// Mitsubishi GX Works2 project: SEMAFARO   PLC: Q03UDV

PROGRAM MAIN
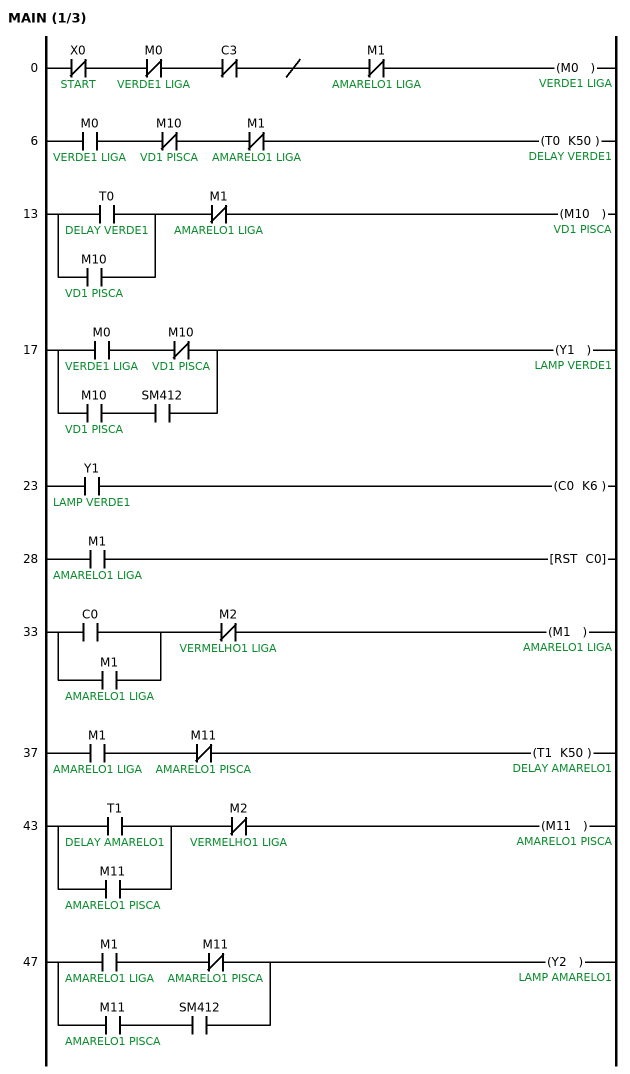
0     LDI     X0  ; START
      ANI     M0  ; VERDE1 LIGA
      ANI     C3
      INV
      ANI     M1  ; AMARELO1 LIGA
      OUT     M0  ; VERDE1 LIGA
6     LD      M0  ; VERDE1 LIGA
      ANI     M10  ; VD1 PISCA
      ANI     M1  ; AMARELO1 LIGA
      OUT     T0 K50  ; DELAY VERDE1
13    LD      T0  ; DELAY VERDE1
      OR      M10  ; VD1 PISCA
      ANI     M1  ; AMARELO1 LIGA
      OUT     M10  ; VD1 PISCA
17    LD      M0  ; VERDE1 LIGA
      ANI     M10  ; VD1 PISCA
      LD      M10  ; VD1 PISCA
      AND     SM412
      ORB
      OUT     Y1  ; LAMP VERDE1
23    LD      Y1  ; LAMP VERDE1
      OUT     C0 K6
28    LD      M1  ; AMARELO1 LIGA
      RST     C0
33    LD      C0
      OR      M1  ; AMARELO1 LIGA
      ANI     M2  ; VERMELHO1 LIGA
      OUT     M1  ; AMARELO1 LIGA
37    LD      M1  ; AMARELO1 LIGA
      ANI     M11  ; AMARELO1 PISCA
      OUT     T1 K50  ; DELAY AMARELO1
43    LD      T1  ; DELAY AMARELO1
      OR      M11  ; AMARELO1 PISCA
      ANI     M2  ; VERMELHO1 LIGA
      OUT     M11  ; AMARELO1 PISCA
47    LD      M1  ; AMARELO1 LIGA
      ANI     M11  ; AMARELO1 PISCA
      LD      M11  ; AMARELO1 PISCA
      AND     SM412
      ORB
      OUT     Y2  ; LAMP AMARELO1
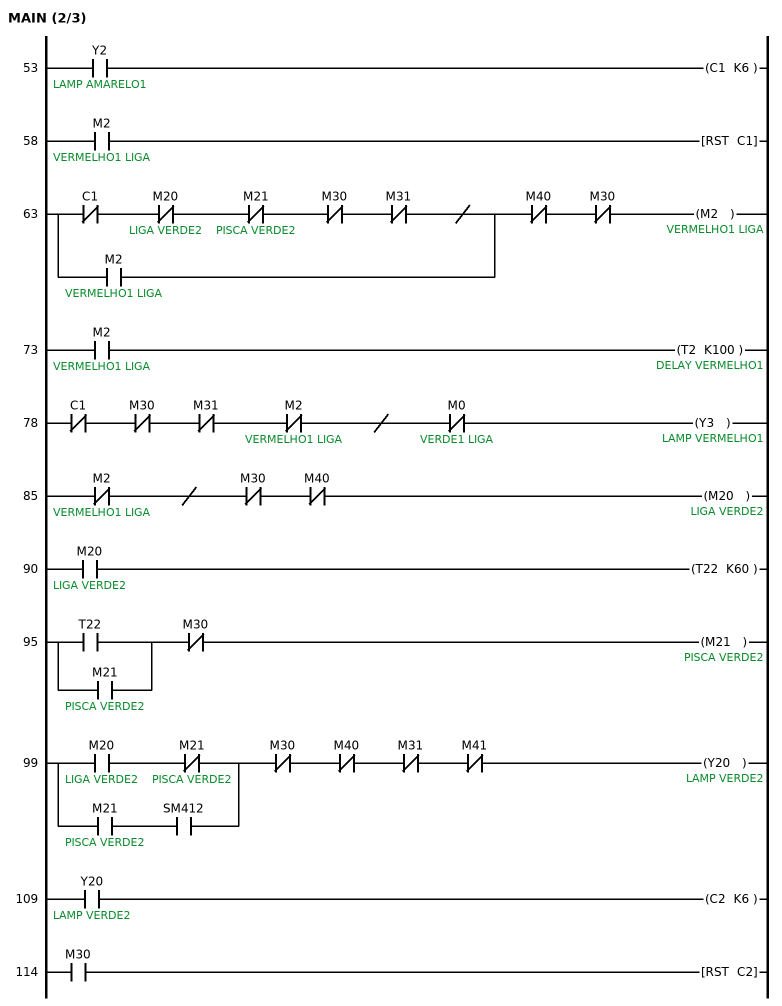
53    LD      Y2  ; LAMP AMARELO1
      OUT     C1 K6
58    LD      M2  ; VERMELHO1 LIGA
      RST     C1
63    LDI     C1
      ANI     M20  ; LIGA VERDE2
      ANI     M21  ; PISCA VERDE2
      ANI     M30
      ANI     M31
      INV
      OR      M2  ; VERMELHO1 LIGA
      ANI     M40
      ANI     M30
      OUT     M2  ; VERMELHO1 LIGA
73    LD      M2  ; VERMELHO1 LIGA
      OUT     T2 K100  ; DELAY VERMELHO1
78    LDI     C1
      ANI     M30
      ANI     M31
      ANI     M2  ; VERMELHO1 LIGA
      INV
      ANI     M0  ; VERDE1 LIGA
      OUT     Y3  ; LAMP VERMELHO1
85    LDI     M2  ; VERMELHO1 LIGA
      INV
      ANI     M30
      ANI     M40
      OUT     M20  ; LIGA VERDE2
90    LD      M20  ; LIGA VERDE2
      OUT     T22 K60
95    LD      T22
      OR      M21  ; PISCA VERDE2
      ANI     M30
      OUT     M21  ; PISCA VERDE2
99    LD      M20  ; LIGA VERDE2
      ANI     M21  ; PISCA VERDE2
      LD      M21  ; PISCA VERDE2
      AND     SM412
      ORB
      ANI     M30
      ANI     M40
      ANI     M31
      ANI     M41
      OUT     Y20  ; LAMP VERDE2
109   LD      Y20  ; LAMP VERDE2
      OUT     C2 K6
114   LD      M30
      RST     C2
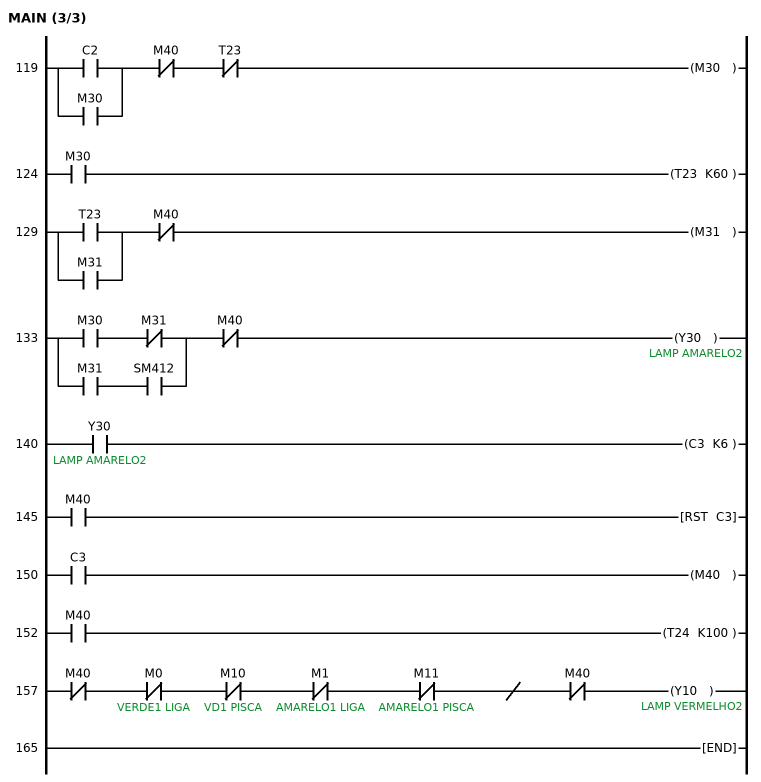
119   LD      C2
      OR      M30
      ANI     M40
      ANI     T23
      OUT     M30
124   LD      M30
      OUT     T23 K60
129   LD      T23
      OR      M31
      ANI     M40
      OUT     M31
133   LD      M30
      ANI     M31
      LD      M31
      AND     SM412
      ORB
      ANI     M40
      OUT     Y30  ; LAMP AMARELO2
140   LD      Y30  ; LAMP AMARELO2
      OUT     C3 K6
145   LD      M40
      RST     C3
150   LD      C3
      OUT     M40
152   LD      M40
      OUT     T24 K100
157   LDI     M40
      ANI     M0  ; VERDE1 LIGA
      ANI     M10  ; VD1 PISCA
      ANI     M1  ; AMARELO1 LIGA
      ANI     M11  ; AMARELO1 PISCA
      INV
      ANI     M40
      OUT     Y10  ; LAMP VERMELHO2
165   END
END_PROGRAM

// device comments not shown above
X1  ; DESLIGAR
Y0  ; verde
